Staubli VAL3: iLevel1.pgx

public program iLevel1(num& nNum[] (dimensions=1))
begin
  nNum=dioGet(iLevel1)
end
